# EPICS autosave request: SPApp/Db/ISCOPumpN_settings.req
#$(P)$(PUMP)PressureSP
#$(P)$(PUMP)FlowRateSP
$(P)$(PUMP)RefillRateSP
$(P)$(PUMP)PressureTweak
$(P)$(PUMP)FlowRateTweak
$(P)$(PUMP)Mode
$(P)$(PUMP)PoorFillAlarm
$(P)$(PUMP)MaxPressureSP
$(P)$(PUMP)MinPressureSP
$(P)$(PUMP)MaxFlowRateSP
$(P)$(PUMP)MaxFlowLimit
$(P)$(PUMP)Description
